# EPICS autosave request: iocBoot/sioc-li20-im01/sioc-li20-im01.req
file "facet2.req" AREA=LI20,POS=1988
file "facet2.req" AREA=LI20,POS=2040
